FUNCTION_BLOCK FB_CuringStationHeaterControl EXTENDS FB_StepperProgram		// This FB is responisble for controlling the heater part of the curing station, we can be in either TEST or WORK mode
VAR_INPUT
	iEstopOk:					BOOL;	// 1 = System is running, no estop pressed
	iEnable:					BOOL;	// When TRUE, this sequence is possible to be run
	iStationId:					UDINT;	// Station nummer, 1..10
	iHeatToTestTemp:			BOOL;	// When TRUE, the test program will run 
	iHeatToWorkTemp:			BOOL;	// When TRUE, will start the heating cycle
	iPt100RawValue:				REAL;	// Raw (unscaled value) of the PT100 element (or any other analog input)
END_VAR
VAR_OUTPUT
	oTestTemperatureReached:	BOOL;	// TRUE when temperature over TEST temperature 
	oWorkTemperatureReached:	BOOL;	// TRUE when temperature over WORK temperature 
	oHeat:						BOOL;	// Heater control
	oFan:						BOOL;	// Fan control
	oTempInC:					REAL;	// Temperature in celcius
	oEnabled:					BOOL;	// When TRUe, the station is enabled
END_VAR
VAR_IN_OUT
	ioHmi:						ST_CURING_STATION_HEATER_CONTROL_HMI;
	ioStaticSettings:			ST_CURING_STATION_HEATER_CONTROL_STATIC_SETTINGS;
END_VAR
VAR
	step:						E_CURING_STATION_HEATER_CONTROL_STEPS;
	service:					ST_CURING_STATION_HEATER_CONTROL_SERVICE;
	ai:							FB_AnalogInput;
//	regularThermostat:			FB_Thermostat;
	specialThermostat:			FB_TimeProportionalThermostat;
	targetTemperature:			REAL;
	
//	staticSettings:				ST_CURING_STATION_HEATER_CONTROL_STATIC_SETTINGS;
END_VAR
VAR_STAT PERSISTENT
//	staticSettings:				ST_CURING_STATION_HEATER_CONTROL_STATIC_SETTINGS;
END_VAR

IF (NOT IING.cycleStart) THEN
	//staticSettings := ioHmi.staticSettings;
	//staticSettings:=ioStaticSettings;
	
//	staticSettings := HEATER_CONTROL_SETTINGS.settings;
END_IF

service := ioHmi.service;

callMeRightBeforeSwitchCase(ADR(step));
CASE step OF
	E_CURING_STATION_HEATER_CONTROL_STEPS.INIT:
		gotoNextStep(iCondition := iEnable AND iHeatToTestTemp, iNextStep := E_CURING_STATION_HEATER_CONTROL_STEPS.HEAT_TO_TEST_TEMP);
		gotoNextStep(iCondition := iEnable AND iHeatToWorkTemp, iNextStep := E_CURING_STATION_HEATER_CONTROL_STEPS.HEAT_TO_WORK_TEMP);
	
	E_CURING_STATION_HEATER_CONTROL_STEPS.HEAT_TO_TEST_TEMP:
		targetTemperature := ioStaticSettings.testTemperature;
		gotoNextStep(iCondition := NOT iEnable OR NOT iHeatToTestTemp, iNextStep := E_CURING_STATION_HEATER_CONTROL_STEPS.INIT);
	
	E_CURING_STATION_HEATER_CONTROL_STEPS.HEAT_TO_WORK_TEMP:
		targetTemperature := ioStaticSettings.workTemperature;
		gotoNextStep(iCondition := NOT iEnable OR NOT iHeatToWorkTemp, iNextStep := E_CURING_STATION_HEATER_CONTROL_STEPS.INIT);

	E_CURING_STATION_HEATER_CONTROL_STEPS.SAFETY_DOWN:
		gotoNextStep(iEstopOk, E_CURING_STATION_HEATER_CONTROL_STEPS.INIT);
ELSE
	step := E_CURING_STATION_HEATER_CONTROL_STEPS.INIT;
END_CASE
callMeRightAfterSwitchCase(TRUE, IING.STRING_BLANK);


// Safety check
IF (NOT iEstopOk) THEN
	gotoNextStep(iCondition := TRUE, iNextStep := E_CURING_STATION_HEATER_CONTROL_STEPS.SAFETY_DOWN);
END_IF

// Analog input
ai(iRawValue := iPt100RawValue, oScaledValue => oTempInC, iDeviceId := iDeviceId, ioHmi := ioHmi.ai);
//oTempInF := 10000;


// Temperature control/thermostat
//regularThermostat(iTargetValue := targetTemperature, iHysteresis := staticSettings.hysteresis, iMeasuredValue := ai.oScaledValue, ioHmi := ioHmi.regularThermostat);

specialThermostat(iHeat := stepInBetween(E_CURING_STATION_HEATER_CONTROL_STEPS.HEAT_TO_TEST_TEMP, E_CURING_STATION_HEATER_CONTROL_STEPS.HEAT_TO_WORK_TEMP), iTargetTemp := targetTemperature, iMeasuredTemp := ai.oScaledValue,
	iOptionalStartDelay := ULINT_TO_TIME(TIME_TO_ULINT(ioStaticSettings.cycleTime) / ioStaticSettings.nrOfStations),
	iPFactor := ioStaticSettings.pFactor, iMinPowerProcent := ioStaticSettings.minPowerProcent, iMaxPowerProcent := ioStaticSettings.maxPowerProcent, iCycleTime := ioStaticSettings.cycleTime, 
	ioHmi := iohmi.specialThermostat
);

// Controlling of actual outputs
oHeat := iEstopOk AND specialThermostat.oHeat;

// Fan follows the heating element
oFan := oHeat;


oTestTemperatureReached := FC_WithinRange(iTarget := ioStaticSettings.testTemperature, iValue := ai.oScaledValue, iRange := ioStaticSettings.hysteresis);
oWorkTemperatureReached := FC_WithinRange(iTarget := ioStaticSettings.workTemperature, iValue := ai.oScaledValue, iRange := ioStaticSettings.hysteresis);

oEnabled := iEnable;

mStatistics();

mHmi();

METHOD PRIVATE mHmi
{warning disable C0371}
IF (NOT __ISVALIDREF (ioHmi)) THEN
	RETURN;
END_IF

//ioHmi.staticSettings := staticSettings;
ioHmi.service := service;

ioHmi.state.enabled := oEnabled;
ioHmi.state.heat := oHeat;
ioHmi.state.fan := oFan;
ioHmi.state.tempInC := oTempInC;
//ioHmi.state.tempInF := oTempInF;


ioHmi.state.testTemperatureReached := oTestTemperatureReached;
ioHmi.state.workTemperatureReached := oWorkTemperatureReached;

ioHmi.state.stationId := iStationId;


{warning restore C0371}
END_METHOD

METHOD mStatistics : BOOL
VAR_INST
	switchHeatOnCount:		FB_EventCounter;
	heatDurationOnCount:	FB_DurationCounter;
END_VAR
switchHeatOnCount(iEvent := oHeat);

heatDurationOnCount(iSignal := oHeat);
END_METHOD

METHOD PUBLIC stepAsString : T_SHORT_STR
stepAsString := TO_STRING(step);
END_METHOD

END_FUNCTION_BLOCK

(* stored: Version 1.1.0.1
   POU FB_CuringStationHeaterControl: Id {1ce5d6ad-b230-4410-8f4a-6d54ab7fcaf5}, SpecialFunc None
   Method mHmi: Id {3eb1f708-8b61-447b-b9e0-094aa60a8f66}
   Method mStatistics: Id {e508fd74-f26d-4db4-a41a-26505d0db198}
   Method stepAsString: Id {21b3ac32-019d-4399-9b0d-ab8c92392b32} *)
